// TIA Portal V17 export
// export: Created 2024-09-02T12:50:36.0238679Z, ExportSetting WithDefaults, DisplayName Totally Integrated Automation Portal, DisplayVersion V17, DisplayName TIA Portal Openness, DisplayVersion V17, DisplayName TIA Portal Version Control Interface, DisplayVersion V17, DisplayName STEP 7 Professional, DisplayVersion V17, DisplayName STEP 7 Safety, DisplayVersion V17, DisplayName WinCC Professional, DisplayVersion V17
TYPE "TypeMobyAnbauteil_1"
// stored: IsFailsafeCompliant false
   STRUCT
      BauteilTyp : Array[1..11] of Char;   // Typskennzeichnung / Type designation
      BauteilHS : Array[1..3] of Char;   // Herstellernummer / manufacturer's number
      ErsteZeichenHS : Byte;   // Position des ersten Zeichens HerstellerNr / Position of the first character ManufacturerNr
      ErsteZeichenTyp : Byte;   // Position des ersten Zeichens TypNr / Position of the first character TypeNr
      LaengeTyp : Byte;   // Zeichenlaenge des Typs / Character length of type
      LaengeDMC : Byte;   // Zeichenlaenge DMC gesamt / Total character length DMC
   END_STRUCT;
END_TYPE
